TYPE ST_Enclosureclimate_events :
STRUCT
	b_HumidityHigh 			: BOOL;
	b_HumidityTooHigh 		: BOOL;
	b_TemperatureHigh		: BOOL;
	b_TemperatureTooHigh	: BOOL;
	b_TemperatureLow		: BOOL;
	b_TemperatureTooLow		: BOOL;
	b_AIOverrange			: BOOL;
	b_AIUnderrange			: BOOL;
	b_AIError				: BOOL;
	b_DewpointTooHigh		: BOOL;
END_STRUCT
END_TYPE

(* stored: Version 1.1.0.1, ProductVersion 3.1.4026.18
   DUT ST_Enclosureclimate_events: Id {a14bd982-fb45-435e-86f6-c090f96fd5de} *)
